(* Logix 5000 project; controller CIP_Server 1769-L16ER-BB1B rev 32.11; software revision 32.00 *)

TASK MainTask (continuous, watchdog 500 ms) : MainProgram

MODULES
   Local : 1769-L16ER-BB1B (PointIO 0, rev 32.11)
      Discrete_IO : Embedded (PointIO 1, rev 32.11, Output RPI 20 ms)
END_MODULES

TYPE ST_CIP_COMS :
STRUCT
   _REAL : REAL;
   _STRING : STRING;
   _INT : INT;
   _DINT : DINT;
   _ArrayREAL : REAL[3];
   _ArraySTRING : STRING[3];
   _ArrayINT : INT[3];
   _ArrayDINT : DINT[3];
END_STRUCT
END_TYPE

VAR_GLOBAL   (* controller tags *)
   Inputs : ST_CIP_COMS := (_REAL := 3.0, _STRING := 'Simple Example:0', _INT := 1, _DINT := 1);
   Outputs : ST_CIP_COMS := (_REAL := 1.9);
END_VAR

PROGRAM MainProgram

ROUTINE MainRoutine   (* ladder *)
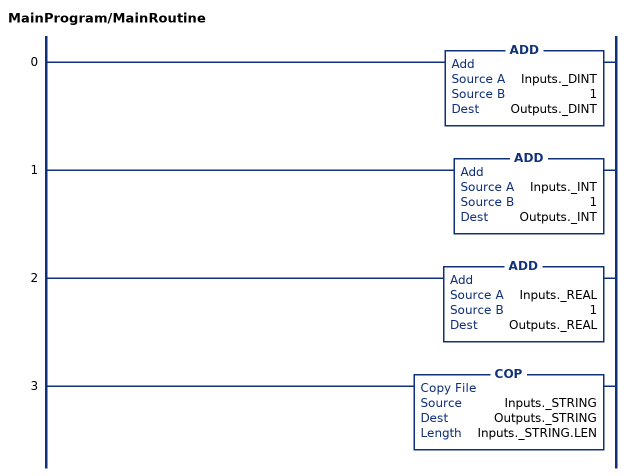
   0: ADD(Inputs._DINT,1,Outputs._DINT);
   1: ADD(Inputs._INT,1,Outputs._INT);
   2: ADD(Inputs._REAL,1,Outputs._REAL);
   3: COP(Inputs._STRING,Outputs._STRING,Inputs._STRING.LEN);
END_ROUTINE
END_PROGRAM
